(* Logix 5000 project; controller Analog_Input Emulate 5570 rev 33.11; software revision 33.00 *)

TASK MainTask (continuous, watchdog 500 ms) : MainProgram, Emulation

MODULES
   Local : Emulate 5570 (ICP 2, rev 33.11)
       : 1756-IB16 (ICP 3, rev 3.1, Input RPI 20 ms)
       : vendor 1 type 7 code 16 (ICP 4, rev 3.1, Output RPI 20 ms)
       : 1756-IF8 (ICP 5, rev 1.1, Input RPI 100 ms)
END_MODULES

PROGRAM Emulation   (* main routine Emulate *)
VAR
   emAIN_RESET : TIMER := (PRE := 3000);
   emCOUNT : COUNTER := (PRE := 6);
   emCOUNT_PULSE : TIMER := (PRE := 6000);
   emPART_A : BOOL;
   emPART_B : BOOL;
END_VAR

ROUTINE Emulate   (* ladder *)
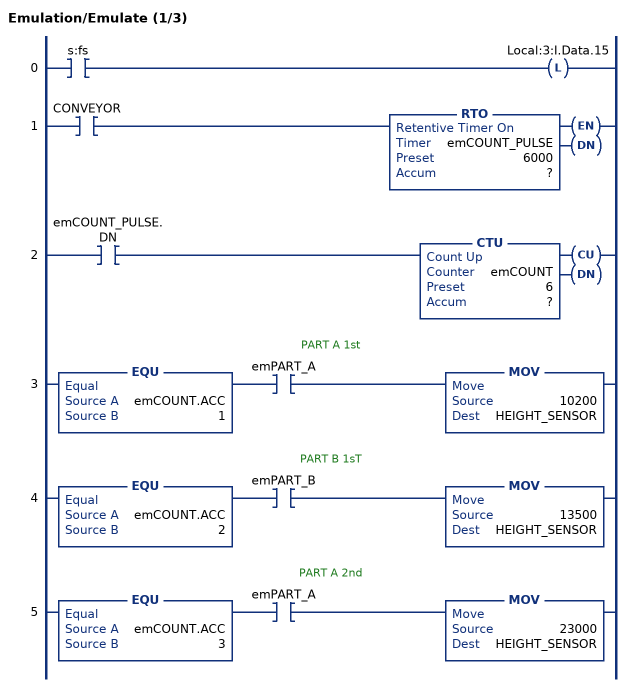
   0: XIC(s:fs)OTL(Local:3:I.Data.15);
   1: XIC(CONVEYOR)RTO(emCOUNT_PULSE,?,?);
   2: XIC(emCOUNT_PULSE.DN)CTU(emCOUNT,?,?);
   // PART A 1st
   3: EQU(emCOUNT.ACC,1)XIC(emPART_A)MOV(10200,HEIGHT_SENSOR);
   // PART B 1sT
   4: EQU(emCOUNT.ACC,2)XIC(emPART_B)MOV(13500,HEIGHT_SENSOR);
   // PART A 2nd
   5: EQU(emCOUNT.ACC,3)XIC(emPART_A)MOV(23000,HEIGHT_SENSOR);
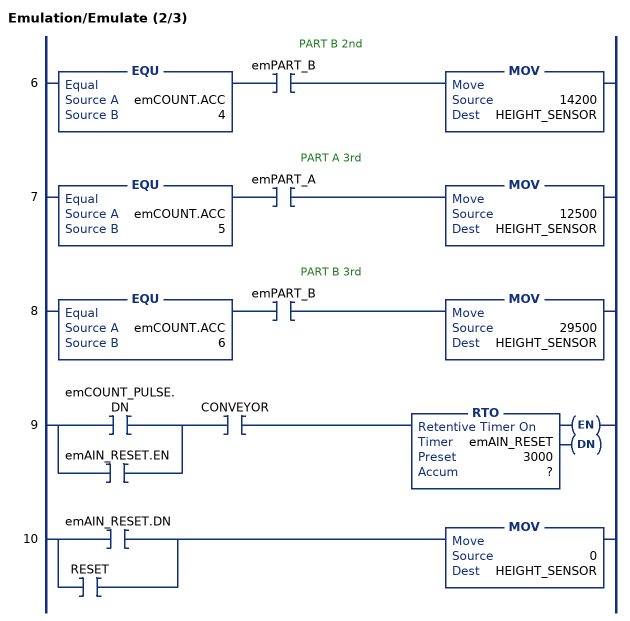
   // PART B 2nd
   6: EQU(emCOUNT.ACC,4)XIC(emPART_B)MOV(14200,HEIGHT_SENSOR);
   // PART A 3rd
   7: EQU(emCOUNT.ACC,5)XIC(emPART_A)MOV(12500,HEIGHT_SENSOR);
   // PART B 3rd
   8: EQU(emCOUNT.ACC,6)XIC(emPART_B)MOV(29500,HEIGHT_SENSOR);
   9: [XIC(emCOUNT_PULSE.DN) ,XIC(emAIN_RESET.EN) ]XIC(CONVEYOR)RTO(emAIN_RESET,?,?);
   10: [XIC(emAIN_RESET.DN) ,XIC(RESET) ]MOV(0,HEIGHT_SENSOR);
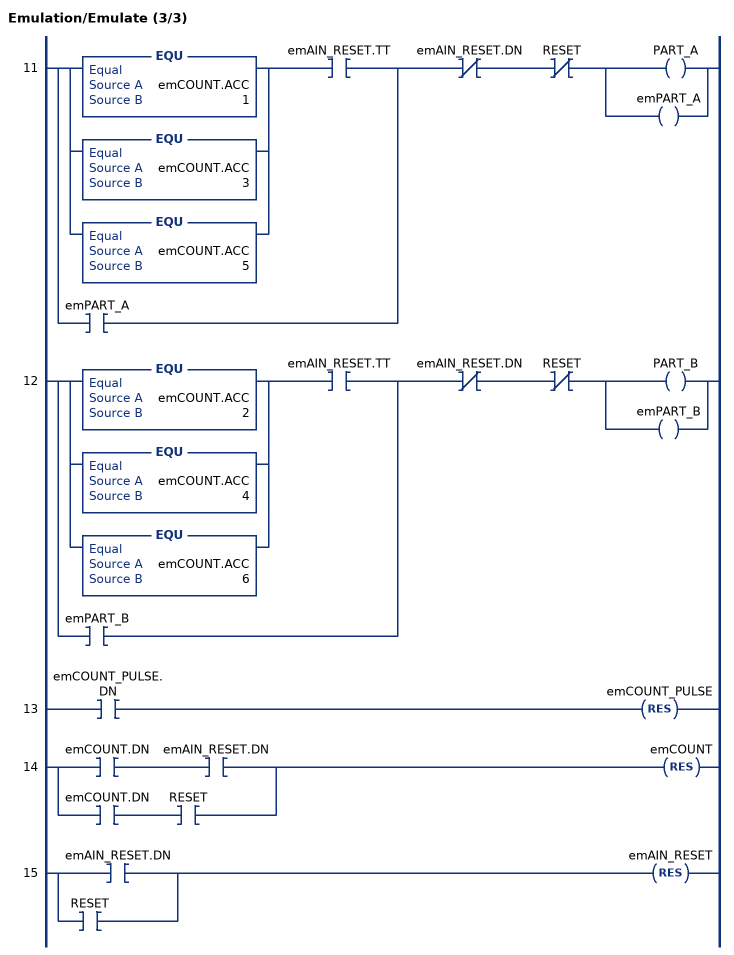
   11: [[EQU(emCOUNT.ACC,1) ,EQU(emCOUNT.ACC,3) ,EQU(emCOUNT.ACC,5) ] XIC(emAIN_RESET.TT) ,XIC(emPART_A) ]XIO(emAIN_RESET.DN)XIO(RESET)[OTE(PART_A) ,OTE(emPART_A) ];
   12: [[EQU(emCOUNT.ACC,2) ,EQU(emCOUNT.ACC,4) ,EQU(emCOUNT.ACC,6) ] XIC(emAIN_RESET.TT) ,XIC(emPART_B) ]XIO(emAIN_RESET.DN)XIO(RESET)[OTE(PART_B) ,OTE(emPART_B) ];
   13: XIC(emCOUNT_PULSE.DN)RES(emCOUNT_PULSE);
   14: [XIC(emCOUNT.DN) XIC(emAIN_RESET.DN) ,XIC(emCOUNT.DN) XIC(RESET) ]RES(emCOUNT);
   15: [XIC(emAIN_RESET.DN) ,XIC(RESET) ]RES(emAIN_RESET);
END_ROUTINE
END_PROGRAM

PROGRAM MainProgram   (* main routine MainRoutine *)

ROUTINE MainRoutine   (* ladder *)
   0: ;
END_ROUTINE
END_PROGRAM
